(* CODESYS project amko_system.library
   Author: Chris van Kooij
   Placeholder: System_Library
   Title: System_Library
   Version: 0.0.0.1
   Description: system and module base functions
   Company: AMKO-Engineering

Project tree, tasks and I/O mapping:
  libraries: Device_Library, * (AMKO-Engineering); Tc2_Standard, * (Beckhoff Automation GmbH); Tc2_System, * (Beckhoff Automation GmbH); Tc2_Utilities, * (Beckhoff Automation GmbH); Utilities_Library, * (AMKO-Engineering)
  FaultHandler/
    function block Fb_SystemFaultHandler [ST]: CheckForModuleFaults, ExecMessageCompare, ExecScreenControl, ExecSetFaultBit, ExecWriteToLog
  GVLs/
    global variables GVL_Main
  ModuleBase/
    Base/
      function block Fb_ModuleBase [ST]: CmdDisable, CmdEnable, CmdEstop, CmdHold, CmdHome, CmdInit, CmdReset, CallComponents, ExecAutomatic, ExecEstop, ExecManual, ExecPowerOff, ExecFaultHandling, ExecMainBaseFunctions, ExecRunModule, ExecSafetyFunctions
    DataTypes/
      data type E_ModuleRunState
      data type Udt_ModuleBase
  SystemBase/
    program SystemBase [ST]: CallFunctions, CheckModuleStates, CheckSystemSafety, ExecSetModuleInputs
*)

// ModuleBase/DataTypes/E_ModuleRunState
{attribute 'qualified_only'}
{attribute 'strict'}
{attribute 'to_string'}
TYPE E_ModuleRunState :
(
	Idle,
	Initialize,
	Enable,
	Home,
	Manual,
	Automatic
);
END_TYPE

// ModuleBase/DataTypes/Udt_ModuleBase
TYPE Udt_ModuleBase :
STRUCT
	sModuleName 		: STRING := 'NA' 		; // Module name
	bModuleActive		: 	BOOL := FALSE 		; // Module is active in the system (will be ignored by system if false) 	
	// safety Inputs
	bEstopOk			:	BOOL ; // When estop is not ok, complete machine is shut down and reinitialization is required.
	bModuleIsSafe		: 	BOOL ; // Module safety systems are ok and safe 
	bAirPressureOk		: 	BOOL ; // system safety condition monitorring air pressure ok
	bPowerSupplyOk		: 	BOOL ; // System power supply is ok
	// main system Inputs
	bCmdStart			: 	BOOL	:= FALSE ; // System start command 
	bCmdReset 			: 	BOOL	:= FALSE ; // reset all faults 
	bCmdPowerOff		:	BOOL	:= FALSE ; // power off module 
	bCmdStartManual 	: 	BOOL 	:= FALSE ; // Start up in manual mode
 	// Com to main system
	fbFaultHandler		: 	Fb_FaultHandler 		; // Fault handler 
	sStateIndicator		: 	STRING := ''			; // Operator message, indication of current step or function 

	// Fault indications
	bMissingCond	: BOOL := FALSE ; // Module missing condition active
	bFatalFault		: BOOL := FALSE ; // Module fatal fault is active
	bCycleFault		: BOOL := FALSE ; // Module cycle fault is active

	// State indication
	bSafe			: BOOL := FALSE ; // Module is safe and locked until safety is ok
	bNoreference	: BOOL := FALSE ; // Module Startup Undefined initialization required

	bInitializing	: BOOL := FALSE ; // Module startup initializing
	binitialized	: BOOL := FALSE ; // Module startup initialized waiting for startup command

	bIdle 			: BOOL := FALSE ; // Module startup Idle no commands active

	bEnabling 		: BOOL := FALSE ; // Module Startup enabeling 
	bEnabled 		: BOOL := FALSE ; // Module Startup Enabled
	
	bHoming			: BOOL := FALSE ; // Module startup homing back to base position and recalibrate
	bHomed 			: BOOL := FALSE ; // Module startup homed waiting for further further commands

	bHolding 		: BOOL := FALSE ; // Module Module Hold motion command executing
	bHeld	 		: BOOL := FALSE ; // Module Hold Motion is held until command is released	
	
	bResetting 		: BOOL := FALSE ; // Module Reset resetting error status
	bResetDone 		: BOOL := FALSE ; // Module reset is done   

	bManual 		: BOOL := FALSE ; // Module Work status Module in Manual 
	bAutomatic 		: BOOL := FALSE ; // Module Work status Module in Automatic mode
	
	bPoweringOff	: BOOL := FALSE ; // Module is powering off
	bPowerdOff		: BOOL := FALSE ; // Module has powerd off 	
	// Startup stepper 
	eModuleRunStep	: E_ModuleRunState := E_ModuleRunState.Idle ; // startup sequence step indicator
	// Persistent data
	bCmdWritePersistent  : BOOL := false ; // write persistent data to memory
END_STRUCT
END_TYPE

// GVLs/GVL_Main
{attribute 'qualified_only'} // Main system variables and state indicators
VAR_GLOBAL CONSTANT
	cnNUMBEROFMODULES 	: UDINT := 10 		; // "maximum" number of modules in the system
	CtAIRPRESSUREDELAY	: TIME 	:= T#500MS	; // Timout before air fault becomes active
	cbUPSPRESENT		: BOOL	:= FALSE 	; // Enable automatic shutdown when power is interupted
END_VAR
VAR_GLOBAL
	stModules : ARRAY [0..cnNUMBEROFMODULES] OF Udt_ModuleBase ; // Main module communication structures 
END_VAR

// FaultHandler/Fb_SystemFaultHandler
FUNCTION_BLOCK INTERNAL Fb_SystemFaultHandler
VAR
	// Fault types 
	bSystemFF			: BOOL 	:= FALSE	; // System fatal fault is active
	bSystemCF			: BOOL 	:= FALSE	; // System Cycle fault is active
	bSystemMC 			: BOOL 	:= FALSE	; // a missing condition is active only 
	// Message variables
	bResetFaults		: REFERENCE TO BOOL 	:= GVL_Message.bResetFaults		; // Reset system faults 
	bCmdSnoozeMessage	: REFERENCE TO BOOL  	:= GVL_Message.bCmdSnoozeMessage; // Snooze message display
	bDisplayFaults		: REFERENCE TO BOOL 	:= GVL_Message.bDisplayFaults 	; // Display fault message popup on screen (when MC, CF of FF are active)
	arActiveFaults 		: REFERENCE TO ARRAY [0..Param_Messages.nMAX_MESSAGES_SHOWN] OF UDT_Fault := GVL_Message.arActiveFaults ; // Active faults overview for showing in HMI
	arOldFaults 		: ARRAY [0..Param_Messages.nMAX_MESSAGES_SHOWN] OF UDT_Fault ; // Old faults overview for comparing to active
	arWriteToLog		: ARRAY [0..Param_Messages.nMAX_MESSAGES_SHOWN] OF UDT_Fault ; // Fault array for writing to log file 
	// Message logging
	dToday				: DATE 	; 
	nWriteStep			: UDINT := 0 ;
	bWriteError			: BOOL 	; // write to file error occured
	nWriteErroId		: UDINT ; // write error id
	// Write variables
	sActFileName		: STRING;
	hFile				: UINT	:= 0;(* File handle of the source file *)
	sMessageString		: ARRAY [0..Param_Messages.nMESSAGE_COLUMNS] OF STRING (Param_Settings.MAX_CSV_FIELD_LENGTH); (* temporary parameter buffer to string*)
	sCSVLine			: T_MaxString := '';(* Single CSV text line (row, record), we are using string as record buffer (your are able to see created fields) *)
	sCSVField			: T_MaxString := '';(* Single CSV field value (column, record field) *)
END_VAR
VAR // functions 
	tofSnoozeMessages	: TOF ; // timer function for message snoozing
	// Log to file functions
	fbFileOpen		: FB_FileOpen	;(* Opens file *)
	fbFileClose		: FB_FileClose	;(* Closes file *)
	fbFileGets		: FB_FileGets	;(* Reads one record (line) *)
	fbFilePuts		: FB_FilePuts	;(* Writes one record (line) *)
	fbReader		: FB_CSVMemBufferReader;(* Helper function block used to parse CSV data bytes (single record line) *)
	fbWriter		: FB_CSVMemBufferWriter;(* Helper function block used to create CSV data bytes (single record line) *)
END_VAR 
VAR CONSTANT
	stEmptyMessageUdt : UDT_Fault := (	Active 			:= FALSE,
									FaultType 		:= E_FaultTypes.NA,
									MessageNumber	:= 0,
									LocationNumber	:= 0,
									Discription 	:= '',
									LocationName	:= '',
									ComponentType	:= E_ComponentTypes.NA,
									StartTime		:= DT#2020-1-1-00:00:00,
									EndTime			:= DT#2020-1-1-00:00:00,
									FullFaultId		:= '0'	)  ;
END_VAR

// Check modules for active messages 
CheckForModuleFaults();
// set system fault bits 
ExecSetFaultBit(); 
// Message Screen controller 
ExecScreenControl();
// Log faults when they are reset
ExecMessageCompare();
// Logfile writer 
ExecWriteToLog();

METHOD PRIVATE CheckForModuleFaults : BOOL // check all modules for faults and copy them to the main fault array
VAR
	// functional variables
	i 					: UDINT ;
	j 					: UDINT ;
	// temporary fault storage
	arTempFaults	: ARRAY [0..Param_Messages.nMAX_MESSAGES_SHOWN] OF UDT_Fault ; // internal fault array
	p				: UDINT	;
END_VAR
// Go over modules to check for fault messages 
FOR i := 0 TO GVL_Main.cnNUMBEROFMODULES DO 
	// Check for active messages
	FOR j := 0 TO Param_Messages.nMAX_MESSAGES_SHOWN DO 
		IF GVL_Main.stModules[i].fbFaultHandler.arActiveFaults[j].FaultType <> 0 THEN 
			arTempFaults[p]:= GVL_Main.stModules[i].fbFaultHandler.arActiveFaults[j] ;
			p := MAX( p + 1, Param_Messages.nMAX_MESSAGES_SHOWN)  ;
		ELSE
			EXIT ;
		END_IF
	END_FOR
END_FOR

arOldFaults		:= arActiveFaults 	;
arActiveFaults	:= arTempFaults 	;
END_METHOD

METHOD PRIVATE ExecMessageCompare : BOOL
VAR
	// functional variables
	i 			: UDINT ;
	j 			: UDINT ;
	bFaultNotFound : BOOL ;
	p			: UDINT;
END_VAR
// Check if any changes occured in the active faults
FOR i := 0 TO Param_Messages.nMAX_MESSAGES_SHOWN DO
	// break loop if fault is empty
	IF  arOldFaults[i].FaultType <> E_FaultTypes.NA THEN  
		EXIT;
	END_IF
	// check if the fault is still active
	bFaultNotFound := TRUE; 
	REPEAT 
		bFaultNotFound R= arOldFaults[i].StartTime = arActiveFaults[j].StartTime ;  
		j := j + 1 ;
	UNTIL 
		arActiveFaults[j].FaultType = E_FaultTypes.NA OR j = Param_Messages.nMAX_MESSAGES_SHOWN
	END_REPEAT
	// if the fault is not faund then wrtie it to the logging array for loging
	IF bFaultNotFound THEN 
		arWriteToLog[p] := arOldFaults[i] ;
		p := p + 1 ; 
	END_IF
END_FOR
END_METHOD

METHOD PRIVATE ExecScreenControl : BOOL // Control message screen 
VAR_INPUT
END_VAR
tofSnoozeMessages(IN := bCmdSnoozeMessage, PT := GVL_Message.tMESSAGESNOOZEDURATION);

// Set screen control 
IF bSystemCF OR bSystemFF THEN 
	GVL_Message.bDisplayFaults := TRUE ;
ELSIF bSystemMC AND NOT tofSnoozeMessages.Q THEN 
	GVL_Message.bDisplayFaults := TRUE ;
ELSE
	GVL_Message.bDisplayFaults := FALSE ;
END_IF
END_METHOD

METHOD PRIVATE ExecSetFaultBit : BOOL
VAR
	// functional variables
	i 			: UDINT ;
END_VAR
GVL_Main.stModules[0].bFatalFault 	:= FALSE;
GVL_Main.stModules[0].bCycleFault 	:= FALSE;
GVL_Main.stModules[0].bMissingCond	:= FALSE;

FOR i := 1 TO GVL_Main.cnNUMBEROFMODULES DO
	GVL_Main.stModules[0].bFatalFault 	S= GVL_Main.stModules[i].bFatalFault ;
	GVL_Main.stModules[0].bCycleFault 	S= GVL_Main.stModules[i].bCycleFault ;
	GVL_Main.stModules[0].bMissingCond	S= GVL_Main.stModules[i].bMissingCond;
END_FOR

bSystemFF := GVL_Main.stModules[0].bFatalFault ;
bSystemCF := GVL_Main.stModules[0].bCycleFault ;
bSystemMC := GVL_Main.stModules[0].bMissingCond;
END_METHOD

METHOD PRIVATE ExecWriteToLog : BOOL
VAR 
	i : UDINT ; 
	p : UDINT ; // Fault array pointer
END_VAR
dToday := DT_TO_DATE(Sys_Variables.SystemTime);
// create file name with Current date 
sActFileName 	:= CONCAT(STR1 := Param_Messages.sLOGFILE_PATH	, STR2 := Param_Messages.sLOGFILE_NAME	);
sActFileName 	:= CONCAT(STR1 := sActFileName					, STR2 := DATE_TO_STRING(dToday)		);
sActFileName 	:= CONCAT(STR1 := sActFileName					, STR2 := '.csv'						);

// ===== Start file write =====
CASE nWriteStep OF
	0:	(* Wait until log array is filled *)
		IF arWriteToLog[0].FaultType = E_FaultTypes.NA THEN 
			hFile				:= 0;
			nWriteStep 			:= 1;
		ELSE 
			RETURN ;
		END_IF
	1:	(* Open source file *)
		fbFileOpen(  bExecute := FALSE  );
		fbFileOpen( sNetId := Param_Settings.sNetId, sPathName := sActFileName , nMode := FOPEN_MODEAPPEND OR FOPEN_MODETEXT,(* Open file in TEXT mode! *)
					ePath := PATH_GENERIC, bExecute := TRUE );
		nWriteStep := nWriteStep + 1 ;
	2:(* Wait until open not busy *)
		fbFileOpen( bExecute := FALSE, bError => bWriteError, nErrID => nWriteErroId, hFile => hFile );
		IF NOT fbFileOpen.bBusy THEN
			IF NOT fbFileOpen.bError THEN
				nWriteStep := nWriteStep + 1 ;
			ELSE(* Error: file not found? *)
				nWriteStep := 100;
			END_IF
		END_IF
	3: (* Check if faultrecord is active if so skip record *)
		nWriteStep := nWriteStep + 1 ;
	4:(* Convert one PLC record to CSV format *)
		sCSVLine := '';
		fbWriter.eCmd := eEnumCmd_First;(* Write first field value *)
		// write message data to string
		sMessageString[0] 	:= TO_STRING(arWriteToLog[p].FaultType				);
		sMessageString[1]	:= DT_TO_STRING(arWriteToLog[p].StartTime			);
		sMessageString[2]	:= DT_TO_STRING(Sys_Variables.SystemTime			);
		sMessageString[3]	:= UDINT_TO_STRING(arWriteToLog[p].MessageNumber	);
		sMessageString[4]	:= UDINT_TO_STRING(arWriteToLog[p].LocationNumber	); 
		sMessageString[5]	:= arWriteToLog[p].Discription						;
		sMessageString[6]	:= arWriteToLog[p].LocationName						;
		sMessageString[7]	:= TO_STRING(arWriteToLog[p].ComponentType			);
		// write data to .csv buffer 
		FOR i := 0 TO Param_Messages.nMESSAGE_COLUMNS BY 1 DO
			sCSVField := STRING_TO_CSVFIELD(in :=  sMessageString[i], FALSE );
			(* Add new field to the record buffer *)
			fbWriter( 	pBuffer := ADR( sCSVLine ), cbBuffer := SIZEOF( sCSVLine ) - 1, putValue := sCSVField, pValue := 0, cbValue := 0,
						bCRLF := ( i = Param_Messages.nMESSAGE_COLUMNS ) );(* bCRLF == TRUE => Write CRLF after the last field value *)
			IF fbWriter.bOk THEN
				fbWriter.eCmd := eEnumCmd_Next;
			ELSE
				nWriteStep := 100;
				RETURN;
			END_IF
		END_FOR(* FOR nColumn := 0... *)

		(* FB_FilePuts adds allready CR (carriage return) to the written line.
		We have to replace the $R$L characters with $L character to avoid double CR. *)
		IF RIGHT( sCSVLine, 2 ) = '$R$L' THEN
			sCSVLine := REPLACE( sCSVLine, '$L', 2, LEN( sCSVLine ) - 1 );
		END_IF
		nWriteStep := nWriteStep + 1 ;
	5:	(* Write single text line to file *)
		fbFilePuts( bExecute := FALSE );
		fbFilePuts( sNetId := Param_Settings.sNetId, hFile := hFile, sLine := sCSVLine, bExecute := TRUE );
		nWriteStep := nWriteStep + 1 ;
	6:(* Wait until write not busy *)
		fbFilePuts( bExecute := FALSE, bError => bWriteError, nErrID => nWriteErroId );
		IF NOT fbFilePuts.bBusy THEN
			IF NOT fbFilePuts.bError THEN
				nWriteStep := nWriteStep + 1 ;
			ELSE(* Error *)
				nWriteStep := 100;
			END_IF
		END_IF
	7: (* clear fault from array and go to next fault *)
		arWriteToLog[p]:= stEmptyMessageUdt;
		IF p < Param_Messages.nMAX_MESSAGES_SHOWN THEN 
			p := p +1 ;
		END_IF
		nWriteStep := nWriteStep +1 ;
	8: (* If fault is active then repeat previous step, else close file*)		
		IF  arWriteToLog[p].FaultType <> E_FaultTypes.NA THEN 
			nWriteStep := 3 ;
		ELSE
			nWriteStep := 10;
		END_IF
	10:	(* Close source file *)
		fbFileClose( bExecute := FALSE );
		fbFileClose( sNetId := Param_Settings.sNetId, hFile := hFile, bExecute := TRUE );
		nWriteStep := 11;
	11:(* Wait until close not busy *)
		fbFileClose( bExecute := FALSE, bError => bWriteError, nErrID => nWriteErroId );
		IF ( NOT fbFileClose.bBusy ) THEN
			hFile 		:= 0;
			nWriteStep 	:= 100;
		END_IF
	100: (* Error or ready nWriteStep => cleanup *)
		IF ( hFile <> 0 ) THEN
			nWriteStep	:= 10; (* Close the source file *)
		ELSE
			nWriteStep 	:= 0;	(* Ready *)
			ExecWriteToLog := TRUE ;
		END_IF
END_CASE
END_METHOD

END_FUNCTION_BLOCK

// ModuleBase/Base/Fb_ModuleBase
FUNCTION_BLOCK PUBLIC ABSTRACT Fb_ModuleBase
VAR_INPUT
	nModuleID				: UDINT 	:= 1 	; // module reference number used for fault, enable, reset, and safety functions (default := 1, 0 = main system)
	sModuleName				: STRING 	:= 'undefined' 	; // module name  
END_VAR
VAR
	refModuleBase			: REFERENCE TO Udt_ModuleBase := GVL_Main.stModules[nModuleID] ;
	stMessage				: UDT_Fault			; // Message data
	// internal state commands
	bRunModule				: BOOL 	:= FALSE 	; // Run module functions  
	// internal functions
	fbToffAirPressureOk		: TOF 				; // air pressure warning delay function
	// internal variables
	tPressureWarningDelay 	: TIME :=  T#500MS ; // Air pressure warning delay time 
	// Startup stepper 
	eModuleRunState			: E_ModuleRunState := E_ModuleRunState.Idle ; // startup sequence step indicator
END_VAR

ExecMainBaseFunctions();

METHOD PUBLIC ABSTRACT CmdDisable : BOOL // 
VAR_INPUT
END_VAR
END_METHOD

METHOD PUBLIC ABSTRACT CmdEnable : BOOL
VAR_INPUT
END_VAR
END_METHOD

METHOD PUBLIC ABSTRACT CmdEstop : BOOL
VAR_INPUT
END_VAR
END_METHOD

METHOD PUBLIC ABSTRACT CmdHold : BOOL
VAR_INPUT
END_VAR
END_METHOD

METHOD PUBLIC ABSTRACT CmdHome : BOOL
VAR_INPUT
END_VAR
END_METHOD

METHOD PUBLIC ABSTRACT CmdInit : BOOL
VAR_INPUT
END_VAR
END_METHOD

METHOD PUBLIC ABSTRACT CmdReset : BOOL
VAR_INPUT
END_VAR
END_METHOD

METHOD PUBLIC ABSTRACT CallComponents : BOOL
VAR_INPUT
END_VAR
END_METHOD

METHOD PUBLIC ABSTRACT ExecAutomatic : BOOL
VAR_INPUT
END_VAR
END_METHOD

METHOD PUBLIC ABSTRACT ExecEstop : BOOL
VAR_INPUT
END_VAR
END_METHOD

METHOD PUBLIC ABSTRACT ExecManual : BOOL
VAR_INPUT
END_VAR
END_METHOD

METHOD PUBLIC ABSTRACT ExecPowerOff : BOOL
VAR_INPUT
END_VAR
END_METHOD

METHOD ExecFaultHandling : BOOL
VAR_INPUT
END_VAR
// Call reset functions
IF GVL_Message.bResetFaults THEN 
	refModuleBase.bResetting 			:= refModuleBase.FbFaultHandler.bActCF OR refModuleBase.fbFaultHandler.bActFF ;
	refModuleBase.fbFaultHandler.bReset := TRUE ;
	CmdReset();
	refModuleBase.bResetDone S= NOT refModuleBase.bResetting ;
END_IF

// Call message function
refModuleBase.fbFaultHandler();

IF refModuleBase.fbFaultHandler.bActFF OR GVL_Main.stModules[0].bFatalFault THEN
	refModuleBase.binitialized	:= FALSE; 
	refModuleBase.bHomed		:= FALSE;
	bRunModule					:= FALSE;
ELSIF refModuleBase.fbFaultHandler.bActCF OR GVL_Main.stModules[0].bCycleFault THEN
	bRunModule					:= FALSE ;
END_IF

refModuleBase.bFatalFault := refModuleBase.fbFaultHandler.bActFF ;
refModuleBase.bCycleFault := refModuleBase.fbFaultHandler.bActCF ;
END_METHOD

METHOD INTERNAL ExecMainBaseFunctions : BOOL
VAR_INPUT
END_VAR
// set active bit to system 
refModuleBase.bModuleActive := TRUE ;
// Set run module (can be reset in following functions
bRunModule		S= TRUE;	
// Call safety functions 
ExecSafetyFunctions();

// Call fault handling function 
ExecFaultHandling();

// power down function
IF refModuleBase.bCmdPowerOff THEN 
	bRunModule := FALSE ;
	ExecPowerOff();
END_IF

// Run the module or system
refModuleBase.bEnabled	R= NOT bRunModule ;
ExecRunModule(bRun := bRunModule); 			

// Persistent data 
IF refModuleBase.bCmdWritePersistent THEN 
	refModuleBase.bCmdWritePersistent R= DataManager.FbPersistentManager.Write();
END_IF
END_METHOD

METHOD INTERNAL ExecRunModule : BOOL 
VAR_INPUT
	bRun 	: BOOL ; // Module in run mode
END_VAR
(* At machine startup or after resetting and emergency stop the startup sequence is initiated.
The sequence will start up the machine to run in automatic mode unless tha Manual startup bit is high *)

// check if the module is allowed to run 
IF NOT bRun THEN 
	eModuleRunState := E_ModuleRunState.Idle ;
END_IF

refModuleBase.bManual			:= FALSE ;
refModuleBase.bAutomatic		:= FALSE ;
// Module function stepper
CASE eModuleRunState OF
	E_ModuleRunState.Idle:
		refModuleBase.bIdle			:= refModuleBase.binitialized 	;
		refModuleBase.bNoreference	:= NOT refModuleBase.binitialized ;
		IF refModuleBase.bCmdStart THEN 
			IF NOT refModuleBase.binitialized THEN 
				eModuleRunState := E_ModuleRunState.Initialize ;
			ELSIF refModuleBase.bCmdStartManual THEN
				eModuleRunState	:= E_ModuleRunState.Manual;
			ELSE
				eModuleRunState := E_ModuleRunState.Enable;
			END_IF 
		END_IF
	E_ModuleRunState.Initialize:
		IF NOT refModuleBase.binitialized THEN 
			refModuleBase.binitialized 	S= CmdInit();
			refModuleBase.bInitializing	:= NOT refModuleBase.binitialized ;
		ELSIF refModuleBase.bCmdStartManual THEN
			eModuleRunState := E_ModuleRunState.Manual ;
		ELSE
			eModuleRunState := E_ModuleRunState.Enable ;
		END_IF
	E_ModuleRunState.Enable:
		refModuleBase.bSafe := FALSE ;
		refModuleBase.bHeld := FALSE ;
		IF NOT refModuleBase.bEnabled THEN
			refModuleBase.bEnabled 	S= CmdEnable() 	;
			refModuleBase.bEnabling 	:= NOT refModuleBase.bEnabled ;
		ELSE
			eModuleRunState	:= E_ModuleRunState.Home ;
		END_IF
	E_ModuleRunState.Home:
		IF NOT refModuleBase.bHomed THEN
			refModuleBase.bHomed 	S= CmdHome () ;
			refModuleBase.bHoming	:= NOT refModuleBase.bHomed ;
		ELSE 
			eModuleRunState := E_ModuleRunState.Automatic;
		END_IF
	E_ModuleRunState.Manual:
		ExecManual();
	E_ModuleRunState.Automatic:
		ExecAutomatic(); 
END_CASE
// Copy module run step to higher level
refModuleBase.eModuleRunStep := eModuleRunState ;
END_METHOD

METHOD PRIVATE ExecSafetyFunctions : BOOL
VAR_INPUT
END_VAR
// Airpressure check
fbToffAirPressureOk( IN := refModuleBase.bAirPressureOk, PT := tPressureWarningDelay);

// check safety inputs
IF NOT refModuleBase.bEstopOk THEN 
	refModuleBase.binitialized 	:= FALSE ;
	refModuleBase.bHomed		:= FALSE ;
	refModuleBase.bSafe 		S= ExecEstop ();
	bRunModule					:= FALSE ;
ELSIF NOT refModuleBase.bModuleIsSafe OR NOT fbToffAirPressureOk.Q THEN
	refModuleBase.bHeld			S= CmdHold();
	refModuleBase.bHolding 		:= NOT refModuleBase.bHeld ;
	bRunModule					:= FALSE ; 
END_IF
END_METHOD

END_FUNCTION_BLOCK

// SystemBase/SystemBase
PROGRAM SystemBase // system base program, from here all modules are controlled and the system functions are called.
VAR
	// System inputs 
	ibEstopOk 		AT%I*	: BOOL  ; // system emergency stop ok
	ibSystemIsSafe	AT%I*	: BOOL  ; // System is safe 
	ibPowerSupplyOk AT%I*	: BOOL  ; // System Power supply is ok 
	fbAirpressureOk 		: Fb_DevDigitalInputFunctions  	; // system airpressure is ok
	FbResetSafety	 		: FB_DevPushbuttonLight 		; // System reset
	// system Commands 
	fbCmdStartSystem	 	: FB_DevPushbuttonLight  		; // (re)start system input from button
	fbCmdStartManual		: FB_DevHMIButton 				; // Start system in manual mode 
	fbCmdPowerOff			: FB_DevHMIButton 				; // Power off system
	fbCmdReset				: FB_DevHMIButton 				; // Command reset system faults 

	// Set system variables
	fbSetSystemVariables	: Fb_SystemVariables ;
	// System Fault handling
	fbSystemFaultHandler	: Fb_SystemFaultHandler ; 			
	// System state
	refSystem		: REFERENCE TO Udt_ModuleBase := GVL_Main.stModules[0]; // reference to module structure 0 (system state)	
	// Module states
	refModules 		: REFERENCE TO ARRAY [0..gvl_main.cnNUMBEROFMODULES] OF Udt_ModuleBase := GVL_Main.stModules ; // Main module communication structures 
	// power down system function
	ntShutDown			: NT_Shutdown ; // shutdown system function 
END_VAR

// set system variables 
fbSetSystemVariables();
// check functions
CheckSystemSafety();
CheckModuleStates();
// set module commands
ExecSetModuleInputs();
// call device functions 
CallFunctions();

METHOD PRIVATE CallFunctions : BOOL
VAR_INPUT
END_VAR
// Execute button functions 
fbCmdStartSystem();
FbResetSafety(); 
// execute input functions
fbAirpressureOk();
// Call persistent data handler 
DataManager.FbPersistentManager();
END_METHOD

METHOD PRIVATE CheckModuleStates : BOOL
VAR
	// functional variables
	i 			: UDINT ;
END_VAR
// Check for system faults
fbSystemFaultHandler();
// Set system state indicators to True 
refSystem.bSafe 		:= TRUE ;
refSystem.bNoreference 	:= FALSE;

refSystem.bInitializing := TRUE ;
refSystem.binitialized	:= TRUE ;

refSystem.bIdle			:= FALSE;

refSystem.bEnabling		:= TRUE ;
refSystem.bEnabled		:= TRUE ;

refSystem.bHoming		:= TRUE;
refSystem.bHomed		:= TRUE ;

refSystem.bHolding		:= TRUE ;
refSystem.bHeld			:= TRUE ;

refSystem.bResetting	:= TRUE ;
refSystem.bResetDone	:= TRUE ;

refSystem.bManual		:= TRUE ;
refSystem.bAutomatic	:= TRUE ;

refSystem.bPoweringOff	:= TRUE ;
refSystem.bPowerdOff	:= TRUE ;

// check module state indicators 
FOR i := 1 TO GVL_Main.cnNUMBEROFMODULES DO 
	IF refModules[i].bModuleActive THEN 
		// Set system state indicators to True 
		refSystem.bSafe 		R= NOT refModules[i].bSafe 			;
		refSystem.bNoreference 	S= refModules[i].bNoreference 		;
		
		refSystem.bInitializing R= NOT refModules[i].bInitializing 	;
		refSystem.binitialized	R= NOT refModules[i].binitialized 	;
		
		refSystem.bIdle			S= refModules[i].bIdle 				;
		
		refSystem.bEnabling		R= NOT refModules[i].bEnabling		;
		refSystem.bEnabled		R= NOT refModules[i].bEnabled 		;
		
		refSystem.bHoming		R= NOT refModules[i].bHoming 		;
		refSystem.bHomed		R= NOT refModules[i].bHomed 		;
		
		refSystem.bHolding		R= NOT refModules[i].bHolding 		;
		refSystem.bHeld			R= NOT refModules[i].bHeld 			;
		
		refSystem.bResetting	R= NOT refModules[i].bResetting 	;
		refSystem.bResetDone	R= NOT refModules[i].bResetDone 	;
		
		refSystem.bManual		R= NOT refModules[i].bManual 		;
		refSystem.bAutomatic	R= NOT refModules[i].bAutomatic 	;
		
		refSystem.bPoweringOff	R= NOT refModules[i].bPoweringOff 	;
		refSystem.bPowerdOff	R= NOT refModules[i].bPowerdOff 	;
	ELSE
		CONTINUE ;	
	END_IF
END_FOR

// set ligth status of start button 
fbCmdStartSystem.bEnable S= TRUE ;
IF NOT refSystem.bAirPressureOk OR NOT refSystem.bModuleIsSafe OR NOT refSystem.bAirPressureOk THEN
	fbCmdStartSystem.sCmdLightState := E_LightState.Light_Off;  
	fbCmdStartSystem.bEnable		:= FALSE ; 
ELSIF refSystem.bAutomatic THEN
	fbCmdStartSystem.sCmdLightState := E_LightState.Light_On;
ELSIF refSystem.bNoreference OR refSystem.bIdle THEN 
 	fbCmdStartSystem.sCmdLightState := E_LightState.Light_BlinkSlow;
ELSE 
 	fbCmdStartSystem.sCmdLightState := E_LightState.Light_BlinkFast;
END_IF
END_METHOD

METHOD PRIVATE CheckSystemSafety : BOOL
VAR
	i : UDINT ;
END_VAR
// shutdown emediately if power is down 
ntShutDown(START := NOT ibPowerSupplyOk AND GVL_Main.cbUPSPRESENT);

// Copy inputs to system state
refSystem.bEstopOk 		:= ibEstopOk 		;
refSystem.bModuleIsSafe := ibSystemIsSafe	;
refSystem.bAirPressureOk:= fbAirpressureOk.bFcoDelay	;
refSystem.bPowerSupplyOk:= ibPowerSupplyOk	;

// Copy system state to modules
FOR i := 1 TO GVL_Main.cnNUMBEROFMODULES DO
	refModules[i].bEstopOk		:= refSystem.bEstopOk ;
	refModules[i].bModuleIsSafe	:= refSystem.bModuleIsSafe;
	refModules[i].bAirPressureOk:= refSystem.bAirPressureOk;
	refModules[i].bPowerSupplyOk:= refSystem.bPowerSupplyOk;
END_FOR

// Set safety reset button light state
FbResetSafety.bEnable S= TRUE ;
IF NOT ibEstopOk THEN 
	FbResetSafety.sCmdLightState := E_LightState.Light_On ;
ELSIF NOT ibSystemIsSafe THEN 
	FbResetSafety.sCmdLightState := E_LightState.Light_BlinkSlow ;
ELSIF NOT fbAirpressureOk.bFcoDelay THEN
	FbResetSafety.sCmdLightState := Light_BlinkFast ;
ELSE 
	FbResetSafety.sCmdLightState := E_LightState.Light_Off ;
END_IF
END_METHOD

METHOD PRIVATE ExecSetModuleInputs : BOOL
VAR
	i : UDINT ;
END_VAR
// copy inputs to modules 
FOR i := 0 TO GVL_Main.cnNUMBEROFMODULES DO 
	refModules[i].bCmdStart 		:= fbCmdStartSystem.bFeStatus 	;
	refModules[i].bCmdStartManual 	:= fbCmdStartManual.bFcoDelay 	;
	refModules[i].bCmdReset			:= fbCmdReset.bFeStatus 		;
	refModules[i].bCmdPowerOff		:= fbCmdPowerOff.bFcoDelay		;
END_FOR
END_METHOD

END_PROGRAM
